// TwinCAT 3 PLC project PLCstudent
// ProgramVersion: 3.1.4026.20
// libraries:
//   Tc2_Standard, * (Beckhoff Automation GmbH)
//   Tc2_System, * (Beckhoff Automation GmbH)
// project tree:
//   GVLs/ GVL.TcGVL
//   / PlcTask.TcTTO
//   POUs/ FunktionBlockDiagram.TcPOU, MAIN.TcPOU
// real-time tasks:
//   TASK PlcTask: cycle T#10ms, priority 20, ADS port 350
//   TASK PlcTask1: cycle T#10ms, priority 21, ADS port 351
// variable links:
//   PLCsim/PLCsim Instance <-> PLCstudent/PLCstudent Instance
//     PlcTask Inputs/GVL.isStatusText <-> PlcTask Outputs/GVL.qsStatusText
//     PlcTask Inputs/GVL.iwPumpSpeed <-> PlcTask Outputs/GVL.qwPumpSpeed
//     PlcTask Outputs/GVL.qwActualLevel <-> PlcTask Inputs/GVL.iwActualLevel

CONFIGURATION PLCstudent
    RESOURCE PLC ON TwinCAT3
        TASK PlcTask(INTERVAL := T#10ms, PRIORITY := 20);
        PROGRAM MAIN WITH PlcTask : MAIN;
    END_RESOURCE
END_CONFIGURATION

// ---- GVLs/GVL.TcGVL
{attribute 'qualified_only'}
VAR_GLOBAL

	qwPumpSpeed   		AT%Q* :  WORD; 	// Speed of the flow into the tank 0 - 100%
										// 40% slowly drain 50% stand still 60% filling
										

	qsStatusText 		AT%Q* : STRING := 'Test text'; // Text on the info display
	
	iwActualLevel 		AT%I* : WORD;  	// Level in the tank	
	
END_VAR

// ---- POUs/MAIN.TcPOU
PROGRAM MAIN
VAR
    levelInt : INT;
    pumpCalc : INT;
END_VAR


(* On/Off tank control *)

IF GVL.iwActualLevel < 40 THEN
    GVL.qwPumpSpeed := 60;
    GVL.qsStatusText := 'Low level';

ELSIF GVL.iwActualLevel > 60 THEN
    GVL.qwPumpSpeed := 0;
    GVL.qsStatusText := 'High level';

ELSE
    GVL.qwPumpSpeed := 40;
    GVL.qsStatusText := 'Normal level';
END_IF;


(* P controller *)

levelInt := WORD_TO_INT(GVL.iwActualLevel);

pumpCalc := (50 - levelInt) * 10;

IF pumpCalc < 0 THEN
    pumpCalc := 0;
END_IF;

GVL.qwPumpSpeed := INT_TO_WORD(pumpCalc);

END_PROGRAM

// ---- POUs/FunktionBlockDiagram.TcPOU
PROGRAM FunktionBlockDiagram
VAR
	 Level_INT : INT;
	 Error_INT : INT;
	 Pump_INT : INT;
	 Pump_LIMIT: INT;
END_VAR

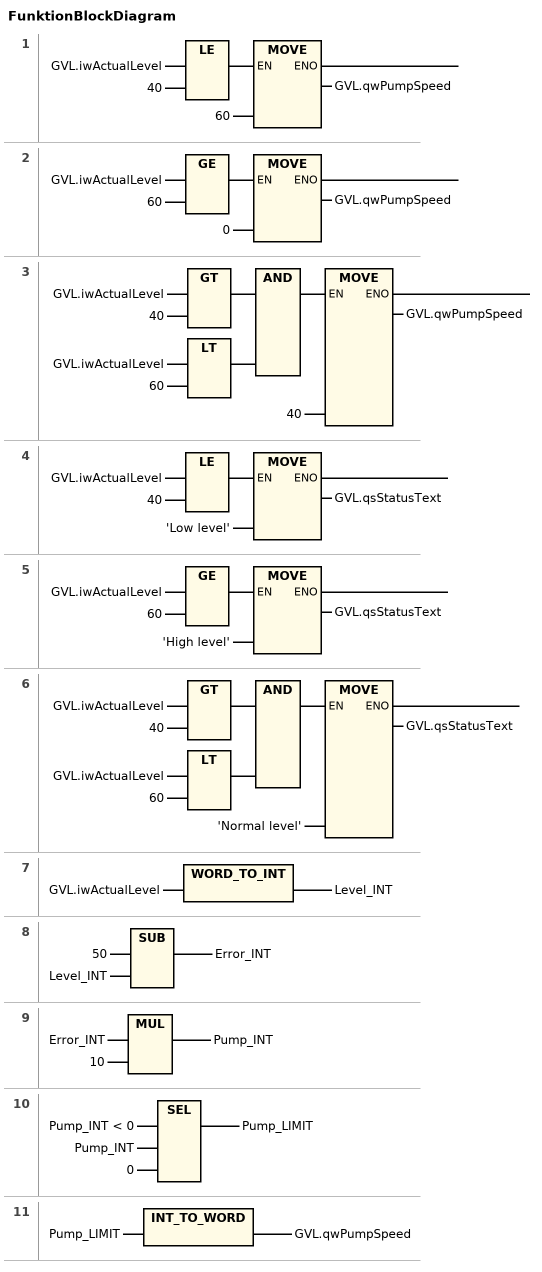
// NETWORK 1
IF GVL.iwActualLevel <= 40 THEN GVL.qwPumpSpeed := 60; END_IF

// NETWORK 2
IF GVL.iwActualLevel >= 60 THEN GVL.qwPumpSpeed := 0; END_IF

// NETWORK 3
IF GVL.iwActualLevel > 40 AND GVL.iwActualLevel < 60 THEN GVL.qwPumpSpeed := 40; END_IF

// NETWORK 4
IF GVL.iwActualLevel <= 40 THEN GVL.qsStatusText := 'Low level'; END_IF

// NETWORK 5
IF GVL.iwActualLevel >= 60 THEN GVL.qsStatusText := 'High level'; END_IF

// NETWORK 6
IF GVL.iwActualLevel > 40 AND GVL.iwActualLevel < 60 THEN GVL.qsStatusText := 'Normal level'; END_IF

// NETWORK 7
Level_INT := WORD_TO_INT(GVL.iwActualLevel);

// NETWORK 8
Error_INT := 50 - Level_INT;

// NETWORK 9
Pump_INT := Error_INT * 10;

// NETWORK 10
Pump_LIMIT := SEL(Pump_INT < 0, Pump_INT, 0);

// NETWORK 11
GVL.qwPumpSpeed := INT_TO_WORD(Pump_LIMIT);

END_PROGRAM
